// TIA Portal V19 export
DATA_BLOCK "Data_block_1"   // DB3
{ S7_Optimized_Access := 'TRUE' }
// stored: MemoryReserve 100
   VAR
      diStart : Bool;
      doDiode : Bool;
   END_VAR
BEGIN
END_DATA_BLOCK
